KUKA KRL data list: ps_ltc_geo_c2.dat

&ACCESS RVO1
&REL 132
&COMMENT GUN C2 geom Accelo
&PARAM DISKPATH = KRC:\R1\Program\SOLDA LTC
DEFDAT  ps_ltc_geo_c2
;FOLD EXTERNAL DECLARATIONS;%{PE}%MKUKATPBASIS,%CEXT,%VCOMMON,%P
;FOLD GRIPPERTECH EXT
EXT  H50 (INT  :IN,INT  :IN,INT  :IN,GRP_TYP  :IN )
;ENDFOLD (GRIPPERTECH EXT)
;FOLD SPOTTECH EXT
EXT  USERSPOT (S_COMMAND  :IN,SPOT_TYPE  :IN )
;ENDFOLD (SPOTTECH EXT)
;FOLD BASISTECH EXT;%{PE}%MKUKATPBASIS,%CEXT,%VEXT,%P
EXT  BAS (BAS_COMMAND  :IN,REAL  :IN )
DECL INT SUCCESS
;ENDFOLD (BASISTECH EXT)
;FOLD USER EXT;%{E}%MKUKATPUSER,%CEXT,%VEXT,%P
;Make your modifications here

;ENDFOLD (USER EXT)
;ENDFOLD (EXTERNAL DECLARATIONS)
;# ============ START PATH : swp_p13050r3_ltc_geo_c2 =============
DECL FDAT Flx828={TOOL_NO 2,BASE_NO 2,IPO_FRAME #BASE,POINT2[] " "}
DECL PDAT PP_OLP7={VEL 100.0,ACC 100.0,APO_DIST 30.0,APO_MODE #CDIS}
DECL E6POS Xlx828={X 1313.89404,Y -1331.46704,Z 523.221985,A -13.1561899,B 25.8715191,C 86.3671722,S 2,T 11,E1 5636.96094,E2 0.0,E3 0.0,E4 0.0,E5 0.0,E6 0.0}
DECL FDAT Flx827={TOOL_NO 2,BASE_NO 2,IPO_FRAME #BASE,POINT2[] " "}
DECL PDAT PP_OLP8={VEL 100.0,ACC 100.0,APO_DIST 30.0,APO_MODE #CDIS}
DECL E6POS Xlx827={X 1268.92896,Y -1028.29199,Z 484.852692,A 0.744642675,B 44.8028793,C 92.9150925,S 2,T 11,E1 5636.54883,E2 0.0,E3 0.0,E4 0.0,E5 0.0,E6 0.0}
DECL FDAT Flx826={TOOL_NO 2,BASE_NO 2,IPO_FRAME #BASE,POINT2[] " "}
DECL PDAT PP_OLP9={VEL 100.0,ACC 100.0,APO_DIST 100.0,APO_MODE #CDIS}
DECL E6POS Xlx826={X 1247.14197,Y -839.330017,Z 487.233398,A 0.873326421,B 46.5667191,C 93.0090027,S 2,T 11,E1 5636.54297,E2 0.0,E3 0.0,E4 0.0,E5 0.0,E6 0.0}
DECL FDAT Fswp_60_0399={TOOL_NO 2,BASE_NO 2,IPO_FRAME #BASE,POINT2[] " "}
DECL PDAT PP_OLP10={VEL 100.0,ACC 100.0,APO_DIST 0.0}
DECL SPOT_TYPE SS_OLP1={GUN 1,PAIR #FIRST,RETR #OPN,CLO_TM 0,PGNO1 1,PRESS1 1.0,PGNO2 0,PRESS2 0.0}
DECL E6POS Xswp_60_0399={X 1474.19995,Y -844.473572,Z 743.300415,A 0.666425526,B -12.8179398,C 91.9345932,S 2,T 11,E1 5636.55713,E2 0.0,E3 0.0,E4 0.0,E5 0.0,E6 0.0}
DECL FDAT Fswp_60_0395={TOOL_NO 2,BASE_NO 2,IPO_FRAME #BASE,POINT2[] " "}
DECL PDAT PP_OLP12={VEL 100.0,ACC 100.0,APO_DIST 0.0}
DECL SPOT_TYPE SS_OLP2={GUN 1,PAIR #FIRST,RETR #OPN,CLO_TM 0,PGNO1 1,PRESS1 1.0,PGNO2 0,PRESS2 0.0}
DECL E6POS Xswp_60_0395={X 1445.07202,Y -842.604614,Z 678.067871,A 1.23996997,B -7.01102686,C 91.9965591,S 2,T 11,E1 5636.50488,E2 0.0,E3 0.0,E4 0.0,E5 0.0,E6 0.0}
DECL FDAT Flx824={TOOL_NO 2,BASE_NO 2,IPO_FRAME #BASE,POINT2[] " "}
DECL PDAT PP_OLP13={VEL 100.0,ACC 100.0,APO_DIST 100.0,APO_MODE #CDIS}
DECL E6POS Xlx824={X 1443.104,Y -839.287109,Z 639.178406,A 2.08833504,B 1.78453195,C 92.0118713,S 2,T 11,E1 5636.50488,E2 0.0,E3 0.0,E4 0.0,E5 0.0,E6 0.0}
DECL FDAT Fswp_60_0393={TOOL_NO 2,BASE_NO 2,IPO_FRAME #BASE,POINT2[] " "}
DECL PDAT PP_OLP14={VEL 100.0,ACC 100.0,APO_DIST 0.0}
DECL SPOT_TYPE SS_OLP3={GUN 1,PAIR #FIRST,RETR #OPN,CLO_TM 0,PGNO1 1,PRESS1 1.0,PGNO2 0,PRESS2 0.0}
DECL E6POS Xswp_60_0393={X 1475.52795,Y -844.253113,Z 638.954773,A -0.0227528196,B 3.38127303,C 92.2101974,S 2,T 11,E1 5636.49512,E2 0.0,E3 0.0,E4 0.0,E5 0.0,E6 0.0}
DECL FDAT Flx823={TOOL_NO 2,BASE_NO 2,IPO_FRAME #BASE,POINT2[] " "}
DECL PDAT PP_OLP16={VEL 100.0,ACC 100.0,APO_DIST 100.0,APO_MODE #CDIS}
DECL E6POS Xlx823={X 1363.30005,Y -822.437317,Z 549.010315,A 0.472675204,B 20.0343704,C 92.5931931,S 2,T 11,E1 5636.54199,E2 0.0,E3 0.0,E4 0.0,E5 0.0,E6 0.0}
DECL FDAT Flx820={TOOL_NO 2,BASE_NO 2,IPO_FRAME #BASE,POINT2[] " "}
DECL PDAT PP_OLP18={VEL 100.0,ACC 100.0,APO_DIST 100.0,APO_MODE #CDIS}
DECL E6POS Xlx820={X 1251.099,Y -1023.78699,Z 483.461304,A 0.771801889,B 44.3958397,C 93.1082611,S 2,T 11,E1 5636.50977,E2 0.0,E3 0.0,E4 0.0,E5 0.0,E6 0.0}
DECL FDAT Flx819={TOOL_NO 2,BASE_NO 2,IPO_FRAME #BASE,POINT2[] " "}
DECL PDAT PP_OLP19={VEL 100.0,ACC 100.0,APO_DIST 100.0,APO_MODE #CDIS}
DECL E6POS Xlx819={X 1444.45801,Y -1414.67004,Z 462.043915,A -12.3754196,B 44.4594803,C 91.9307175,S 2,T 11,E1 5636.50586,E2 0.0,E3 0.0,E4 0.0,E5 0.0,E6 0.0}
DECL FDAT Fswp_60_0341={TOOL_NO 2,BASE_NO 2,IPO_FRAME #BASE,POINT2[] " "}
DECL PDAT PP_OLP21={VEL 100.0,ACC 100.0,APO_DIST 0.0}
DECL SPOT_TYPE SS_OLP4={GUN 1,PAIR #FIRST,RETR #OPN,CLO_TM 0,PGNO1 1,PRESS1 1.0,PGNO2 0,PRESS2 0.0}
DECL E6POS Xswp_60_0341={X 1400.88696,Y -841.813171,Z 60.6647987,A -3.50004601,B 32.0640984,C 89.0238266,S 2,T 11,E1 5553.2959,E2 0.0,E3 0.0,E4 0.0,E5 0.0,E6 0.0}
DECL FDAT Fswp_60_0333={TOOL_NO 2,BASE_NO 2,IPO_FRAME #BASE,POINT2[] " "}
DECL PDAT PP_OLP22={VEL 100.0,ACC 100.0,APO_DIST 0.0}
DECL SPOT_TYPE SS_OLP5={GUN 1,PAIR #FIRST,RETR #OPN,CLO_TM 0,PGNO1 1,PRESS1 1.0,PGNO2 0,PRESS2 0.0}
DECL E6POS Xswp_60_0333={X 1245.823,Y -840.628174,Z 60.1122894,A -3.49715209,B 31.6406898,C 88.9972,S 2,T 11,E1 5553.13379,E2 0.0,E3 0.0,E4 0.0,E5 0.0,E6 0.0}
DECL FDAT Flx815={TOOL_NO 2,BASE_NO 2,IPO_FRAME #BASE,POINT2[] " "}
DECL PDAT PP_OLP23={VEL 100.0,ACC 100.0,APO_DIST 100.0,APO_MODE #CDIS}
DECL E6POS Xlx815={X 1196.84094,Y -826.712402,Z 159.871796,A -3.81221008,B 31.1064892,C 88.8207474,S 2,T 11,E1 5552.36182,E2 0.0,E3 0.0,E4 0.0,E5 0.0,E6 0.0}
DECL FDAT Flx816={TOOL_NO 2,BASE_NO 2,IPO_FRAME #BASE,POINT2[] " "}
DECL PDAT PP_OLP24={VEL 100.0,ACC 100.0,APO_DIST 30.0,APO_MODE #CDIS}
DECL E6POS Xlx816={X 1198.349,Y -1363.80798,Z 157.276199,A -10.3484898,B 31.0169201,C 86.4901962,S 2,T 11,E1 5539.03516,E2 0.0,E3 0.0,E4 0.0,E5 0.0,E6 0.0}
DECL FDAT Flx814={TOOL_NO 2,BASE_NO 2,IPO_FRAME #BASE,POINT2[] " "}
DECL E6POS Xlx814={X 369.932312,Y -1519.18604,Z -172.970001,A -167.901596,B 57.7843094,C -67.7142334,S 2,T 11,E1 4678.13623,E2 0.0,E3 0.0,E4 0.0,E5 0.0,E6 0.0}
DECL FDAT Flx813={TOOL_NO 2,BASE_NO 2,IPO_FRAME #BASE,POINT2[] " "}
DECL E6POS Xlx813={X 428.942688,Y -806.54657,Z -98.9288864,A 175.669601,B 53.0529213,C -91.0339203,S 2,T 11,E1 4678.10986,E2 0.0,E3 0.0,E4 0.0,E5 0.0,E6 0.0}
DECL FDAT Fswp_60_0255={TOOL_NO 2,BASE_NO 2,IPO_FRAME #BASE,POINT2[] " "}
DECL PDAT PP_OLP30={VEL 100.0,ACC 100.0,APO_DIST 0.0}
DECL SPOT_TYPE SS_OLP6={GUN 1,PAIR #FIRST,RETR #OPN,CLO_TM 0,PGNO1 1,PRESS1 1.0,PGNO2 0,PRESS2 0.0}
DECL E6POS Xswp_60_0255={X 300.463989,Y -853.163086,Z -119.2994,A 175.893997,B 45.7151489,C -93.9277267,S 2,T 11,E1 4678.07178,E2 0.0,E3 0.0,E4 0.0,E5 0.0,E6 0.0}
DECL FDAT Fswp_60_0245={TOOL_NO 2,BASE_NO 2,IPO_FRAME #BASE,POINT2[] " "}
DECL PDAT PP_OLP31={VEL 100.0,ACC 100.0,APO_DIST 0.0}
DECL SPOT_TYPE SS_OLP7={GUN 1,PAIR #FIRST,RETR #OPN,CLO_TM 0,PGNO1 1,PRESS1 1.0,PGNO2 0,PRESS2 0.0}
DECL E6POS Xswp_60_0245={X 236.971893,Y -854.070374,Z -10.8238602,A -179.4767,B 23.06007,C -91.1865311,S 2,T 11,E1 4684.35791,E2 0.0,E3 0.0,E4 0.0,E5 0.0,E6 0.0}
DECL FDAT Fswp_60_0235={TOOL_NO 2,BASE_NO 2,IPO_FRAME #BASE,POINT2[] " "}
DECL PDAT PP_OLP33={VEL 100.0,ACC 100.0,APO_DIST 0.0}
DECL SPOT_TYPE SS_OLP8={GUN 1,PAIR #FIRST,RETR #OPN,CLO_TM 0,PGNO1 1,PRESS1 1.0,PGNO2 0,PRESS2 0.0}
DECL E6POS Xswp_60_0235={X 258.574402,Y -852.900208,Z 151.175507,A -179.494904,B -23.2381096,C -89.6756897,S 2,T 11,E1 4681.46387,E2 0.0,E3 0.0,E4 0.0,E5 0.0,E6 0.0}
DECL FDAT Flx798={TOOL_NO 2,BASE_NO 2,IPO_FRAME #BASE,POINT2[] " "}
DECL PDAT PP_OLP34={VEL 100.0,ACC 100.0,APO_DIST 100.0,APO_MODE #CDIS}
DECL E6POS Xlx798={X 268.457794,Y -793.195618,Z 67.879303,A -179.860504,B 7.61739111,C -89.3985977,S 2,T 11,E1 4683.8208,E2 0.0,E3 0.0,E4 0.0,E5 0.0,E6 0.0}
DECL FDAT Flx799={TOOL_NO 2,BASE_NO 2,IPO_FRAME #BASE,POINT2[] " "}
DECL PDAT PP_OLP35={VEL 100.0,ACC 100.0,APO_DIST 100.0,APO_MODE #CDIS}
DECL E6POS Xlx799={X 345.372589,Y -812.418274,Z -84.5929871,A 176.158905,B 42.65382,C -93.2365875,S 2,T 11,E1 4677.79199,E2 0.0,E3 0.0,E4 0.0,E5 0.0,E6 0.0}
DECL FDAT Flx800={TOOL_NO 2,BASE_NO 2,IPO_FRAME #BASE,POINT2[] " "}
DECL E6POS Xlx800={X 428.928711,Y -806.551819,Z -98.9253006,A 175.669693,B 53.0524902,C -91.0339737,S 2,T 11,E1 4686.33398,E2 0.0,E3 0.0,E4 0.0,E5 0.0,E6 0.0}
DECL FDAT Flx802={TOOL_NO 2,BASE_NO 2,IPO_FRAME #BASE,POINT2[] " "}
DECL PDAT PP_OLP37={VEL 100.0,ACC 100.0,APO_DIST 100.0,APO_MODE #CDIS}
DECL E6POS Xlx802={X 410.083588,Y -1114.28699,Z -102.263397,A 175.624405,B 54.5072289,C -91.0710373,S 2,T 11,E1 4684.38477,E2 0.0,E3 0.0,E4 0.0,E5 0.0,E6 0.0}
DECL FDAT Flx801={TOOL_NO 2,BASE_NO 2,IPO_FRAME #BASE,POINT2[] " "}
DECL PDAT PP_OLP38={VEL 100.0,ACC 100.0,APO_DIST 10.0,APO_MODE #CDIS}
DECL E6POS Xlx801={X 350.765411,Y -1468.63098,Z -154.114105,A -172.531601,B 56.018959,C -75.8321533,S 2,T 11,E1 4678.13477,E2 0.0,E3 0.0,E4 0.0,E5 0.0,E6 0.0}
DECL FDAT Flx804={TOOL_NO 2,BASE_NO 2,IPO_FRAME #BASE,POINT2[] " "}
DECL E6POS Xlx804={X 395.674713,Y -813.304382,Z 335.053406,A -179.504196,B 41.2089806,C -87.9716721,S 2,T 11,E1 4687.36084,E2 0.0,E3 0.0,E4 0.0,E5 0.0,E6 0.0}
DECL FDAT Flx803={TOOL_NO 2,BASE_NO 2,IPO_FRAME #BASE,POINT2[] " "}
DECL PDAT PP_OLP45={VEL 100.0,ACC 100.0,APO_DIST 100.0,APO_MODE #CDIS}
DECL E6POS Xlx803={X 236.066498,Y -818.786377,Z 292.583099,A -179.961105,B 26.3373394,C -89.4697876,S 2,T 11,E1 4682.87988,E2 0.0,E3 0.0,E4 0.0,E5 0.0,E6 0.0}
DECL FDAT Fswp_60_0229={TOOL_NO 2,BASE_NO 2,IPO_FRAME #BASE,POINT2[] " ",TQ_STATE FALSE}
DECL PDAT PP_OLP46={VEL 100.0,ACC 100.0,APO_DIST 0.0}
DECL SPOT_TYPE SS_OLP9={GUN 1,PAIR #FIRST,RETR #OPN,CLO_TM 0,PGNO1 1,PRESS1 1.0,PGNO2 0,PRESS2 0.0}
DECL E6POS Xswp_60_0229={X 216.704895,Y -869.258728,Z 250.863495,A -179.965103,B 26.5219803,C -89.4639969,S 2,T 11,E1 4685.6792,E2 0.0,E3 0.0,E4 0.0,E5 0.0,E6 0.0}
DECL FDAT Fswp_60_0225={TOOL_NO 2,BASE_NO 2,IPO_FRAME #BASE,POINT2[] " "}
DECL PDAT PP_OLP47={VEL 100.0,ACC 100.0,APO_DIST 0.0}
DECL SPOT_TYPE SS_OLP10={GUN 1,PAIR #FIRST,RETR #OPN,CLO_TM 0,PGNO1 1,PRESS1 1.0,PGNO2 0,PRESS2 0.0}
DECL E6POS Xswp_60_0225={X 210.434692,Y -869.599915,Z 287.652191,A -178.351898,B 25.9884892,C -88.7657318,S 2,T 11,E1 4685.66895,E2 0.0,E3 0.0,E4 0.0,E5 0.0,E6 0.0}
DECL FDAT Fswp_60_0221={TOOL_NO 2,BASE_NO 2,IPO_FRAME #BASE,POINT2[] " "}
DECL PDAT PP_OLP49={VEL 100.0,ACC 100.0,APO_DIST 0.0}
DECL SPOT_TYPE SS_OLP11={GUN 1,PAIR #FIRST,RETR #OPN,CLO_TM 0,PGNO1 1,PRESS1 1.0,PGNO2 0,PRESS2 0.0}
DECL E6POS Xswp_60_0221={X 174.025696,Y -868.362915,Z 329.479706,A -177.526199,B 4.52676916,C -90.1046982,S 2,T 11,E1 4681.50488,E2 0.0,E3 0.0,E4 0.0,E5 0.0,E6 0.0}
DECL FDAT Flx795={TOOL_NO 2,BASE_NO 2,IPO_FRAME #BASE,POINT2[] " "}
DECL PDAT PP_OLP50={VEL 100.0,ACC 100.0,APO_DIST 100.0,APO_MODE #CDIS}
DECL E6POS Xlx795={X 226.200195,Y -837.525085,Z 348.480286,A -178.942001,B 2.25270796,C -89.7577896,S 2,T 11,E1 4678.92383,E2 0.0,E3 0.0,E4 0.0,E5 0.0,E6 0.0}
DECL FDAT Flx796={TOOL_NO 2,BASE_NO 2,IPO_FRAME #BASE,POINT2[] " "}
DECL PDAT PP_OLP51={VEL 100.0,ACC 100.0,APO_DIST 100.0,APO_MODE #CDIS}
DECL E6POS Xlx796={X 263.717407,Y -815.125122,Z 435.898987,A -178.984207,B 0.893851578,C -89.7701492,S 2,T 11,E1 4682.00098,E2 0.0,E3 0.0,E4 0.0,E5 0.0,E6 0.0}
DECL FDAT Fswp_60_0205={TOOL_NO 2,BASE_NO 2,IPO_FRAME #BASE,POINT2[] " "}
DECL PDAT PP_OLP52={VEL 100.0,ACC 100.0,APO_DIST 0.0}
DECL SPOT_TYPE SS_OLP12={GUN 1,PAIR #FIRST,RETR #OPN,CLO_TM 0,PGNO1 1,PRESS1 1.0,PGNO2 0,PRESS2 0.0}
DECL E6POS Xswp_60_0205={X 265.348785,Y -866.557007,Z 493.816589,A -178.943497,B 1.47540104,C -89.7626266,S 2,T 11,E1 4677.98193,E2 0.0,E3 0.0,E4 0.0,E5 0.0,E6 0.0}
DECL FDAT Fswp_60_0209={TOOL_NO 2,BASE_NO 2,IPO_FRAME #BASE,POINT2[] " "}
DECL SPOT_TYPE SS_OLP13={GUN 1,PAIR #FIRST,RETR #OPN,CLO_TM 0,PGNO1 1,PRESS1 1.0,PGNO2 0,PRESS2 0.0}
DECL E6POS Xswp_60_0209={X 198.4814,Y -864.90863,Z 453.328186,A -179.031296,B -7.38044596,C -89.7764587,S 2,T 11,E1 4674.09521,E2 0.0,E3 0.0,E4 0.0,E5 0.0,E6 0.0}
DECL FDAT Fswp_60_0217={TOOL_NO 2,BASE_NO 2,IPO_FRAME #BASE,POINT2[] " "}
DECL SPOT_TYPE SS_OLP14={GUN 1,PAIR #FIRST,RETR #OPN,CLO_TM 0,PGNO1 1,PRESS1 1.0,PGNO2 0,PRESS2 0.0}
DECL E6POS Xswp_60_0217={X 129.435394,Y -861.487915,Z 279.004608,A 17.8512707,B -39.6672592,C 83.1958389,S 2,T 11,E1 4906.23389,E2 0.0,E3 0.0,E4 0.0,E5 0.0,E6 0.0}
DECL FDAT Fswp_60_0219={TOOL_NO 2,BASE_NO 2,IPO_FRAME #BASE,POINT2[] " "}
DECL SPOT_TYPE SS_OLP15={GUN 1,PAIR #FIRST,RETR #OPN,CLO_TM 0,PGNO1 1,PRESS1 1.0,PGNO2 0,PRESS2 0.0}
DECL E6POS Xswp_60_0219={X 132.783798,Y -863.262512,Z 297.808594,A 16.7955704,B -40.7878494,C 86.3009567,S 2,T 11,E1 4905.89502,E2 0.0,E3 0.0,E4 0.0,E5 0.0,E6 0.0}
DECL FDAT Flx780={TOOL_NO 2,BASE_NO 2,IPO_FRAME #BASE,POINT2[] " "}
DECL PDAT PP_OLP71={VEL 100.0,ACC 100.0,APO_DIST 25.0,APO_MODE #CDIS}
DECL E6POS Xlx780={X -536.1073,Y -3036.90088,Z -433.383789,A -103.127502,B 3.39632702,C 10.3325796,S 2,T 11,E1 3967.95703,E2 0.0,E3 0.0,E4 0.0,E5 0.0,E6 0.0}
DECL FDAT Fswp_60_0201={TOOL_NO 2,BASE_NO 2,IPO_FRAME #BASE,POINT2[] " "}
DECL SPOT_TYPE SS_OLP16={GUN 1,PAIR #FIRST,RETR #OPN,CLO_TM 0,PGNO1 1,PRESS1 1.0,PGNO2 0,PRESS2 0.0}
DECL E6POS Xswp_60_0201={X 229.770004,Y -890.145325,Z 555.893982,A -179.049301,B -22.7869892,C -89.742157,S 2,T 11,E1 4680.5332,E2 0.0,E3 0.0,E4 0.0,E5 0.0,E6 0.0}
DECL FDAT Flx767={TOOL_NO 2,BASE_NO 2,IPO_FRAME #BASE,POINT2[] " "}
DECL PDAT PP_OLP81={VEL 100.0,ACC 100.0,APO_DIST 30.0,APO_MODE #CDIS}
DECL E6POS Xlx767={X -4198.59521,Y -2862.68604,Z -364.78479,A 103.820503,B 2.44905901,C -6.20870399,S 2,T 43,E1 1408.61401,E2 0.0,E3 0.0,E4 0.0,E5 0.0,E6 0.0}
DECL BASIS_SUGG_T LAST_BASIS={POINT1[] "PS01010001              ",POINT2[] "PS01010001              ",CP_PARAMS[] "CPDAT0                  ",PTP_PARAMS[] "PDAT0                   ",CONT[] "                        ",CP_VEL[] "2.0                     ",PTP_VEL[] "100                     ",SPL_NAME[] "S0                      "}
DECL E6POS XP2={X -483.254089,Y -2982.05591,Z -402.20639,A -107.179497,B 0.544633925,C 4.32910204,S 2,T 3,E1 4351.56006,E2 0.0,E3 0.0,E4 0.0,E5 0.0,E6 0.0}
DECL FDAT FP2={TOOL_NO 2,BASE_NO 2,IPO_FRAME #BASE,POINT2[] " ",TQ_STATE FALSE}
DECL PDAT PPDAT2={VEL 100.0,ACC 100.0,APO_DIST 30.0,APO_MODE #CDIS}
DECL SPOT_SUGG_T LAST_SPOT={GUN[] "2                       ",RETR_CMD[] "#OPN                    ",CHOISE[] "#FIRST                  ",CLO_TM[] "1                       ",PGNO1[] "252                     ",PRESS1[] "0                       ",PGNO2[] "1                       ",PRESS2[] "0                       ",SPOT_PARAMS[] "NORMAL                  "}
DECL E6POS XP6={X 1279.60999,Y -1373.32605,Z 198.834396,A -9.93967724,B 7.73596001,C 90.3461227,S 2,T 11,E1 5553.88281,E2 0.0,E3 0.0,E4 0.0,E5 0.0,E6 0.0}
DECL FDAT FP6={TOOL_NO 2,BASE_NO 2,IPO_FRAME #BASE,POINT2[] " ",TQ_STATE FALSE}
DECL PDAT PPDAT6={VEL 100.0,ACC 100.0,APO_DIST 30.0,APO_MODE #CDIS}
DECL E6POS XP7={X 1202.75,Y -808.4328,Z 199.5867,A -5.53556919,B 7.68426991,C 92.4831314,S 2,T 11,E1 5553.88184,E2 0.0,E3 0.0,E4 0.0,E5 0.0,E6 0.0}
DECL FDAT FP7={TOOL_NO 2,BASE_NO 2,IPO_FRAME #BASE,POINT2[] " ",TQ_STATE FALSE}
DECL PDAT PPDAT7={VEL 100.0,ACC 100.0,APO_DIST 100.0}
DECL E6POS XP11={X 262.014008,Y -846.799622,Z 144.059601,A -179.474792,B -23.1920395,C -89.2290115,S 2,T 11,E1 4682.82422,E2 0.0,E3 0.0,E4 0.0,E5 0.0,E6 0.0}
DECL FDAT FP11={TOOL_NO 2,BASE_NO 2,IPO_FRAME #BASE,POINT2[] " ",TQ_STATE FALSE}
DECL PDAT PPDAT11={VEL 100.0,ACC 100.0,APO_DIST 10.0,APO_MODE #CDIS}
DECL LDAT LCPDAT1={VEL 2.0,ACC 100.0,APO_DIST 2.0,APO_FAC 50.0,AXIS_VEL 100.0,AXIS_ACC 100.0,ORI_TYP #VAR,CIRC_TYP #BASE,JERK_FAC 50.0,GEAR_JERK 50.0,EXAX_IGN 0}
DECL LDAT LCPDAT5={VEL 2.0,ACC 100.0,APO_DIST 20.0,APO_FAC 50.0,AXIS_VEL 100.0,AXIS_ACC 100.0,ORI_TYP #VAR,CIRC_TYP #BASE,JERK_FAC 50.0,GEAR_JERK 50.0,EXAX_IGN 0}
DECL LDAT LCPDAT8={VEL 2.0,ACC 100.0,APO_DIST 2.0,APO_FAC 50.0,AXIS_VEL 100.0,AXIS_ACC 100.0,ORI_TYP #VAR,CIRC_TYP #BASE,JERK_FAC 50.0,GEAR_JERK 50.0,EXAX_IGN 0}
DECL E6POS XP28={X 680.9328,Y -2572.68799,Z -141.916397,A -67.8898773,B 12.2103901,C 37.8295212,S 2,T 11,E1 4582.3208,E2 0.0,E3 0.0,E4 0.0,E5 0.0,E6 0.0}
DECL FDAT FP28={TOOL_NO 2,BASE_NO 2,IPO_FRAME #BASE,POINT2[] " ",TQ_STATE FALSE}
DECL PDAT PPDAT28={VEL 100.0,ACC 100.0,APO_DIST 100.0,APO_MODE #CDIS}
DECL E6POS XP30={X 1907.59802,Y -7875.57715,Z 2378.80493,A -86.6201935,B -16.2818298,C 91.4838104,S 2,T 11,E1 5636.49512,E2 0.0,E3 0.0,E4 0.0,E5 0.0,E6 0.0}
DECL FDAT FP30={TOOL_NO 2,BASE_NO 0,IPO_FRAME #BASE,POINT2[] " ",TQ_STATE FALSE}
DECL PDAT PPDAT30={VEL 100.0,ACC 100.0,APO_DIST 20.0,APO_MODE #CDIS}
DECL PDAT PPDAT35={VEL 100.0,ACC 100.0,APO_DIST 10.0,APO_MODE #CDIS}
DECL E6POS XP35={X -142.686005,Y -2282.2041,Z 1278.44495,A 13.8204603,B 2.44905901,C -6.20870399,S 2,T 43,E1 1408.61401,E2 0.0,E3 0.0,E4 0.0,E5 0.0,E6 0.0}
DECL FDAT FP35={TOOL_NO 2,BASE_NO 0,IPO_FRAME #BASE,POINT2[] " ",TQ_STATE FALSE}
DECL PDAT PPDAT36={VEL 100.0,ACC 100.0,APO_DIST 5.0,APO_MODE #CDIS}
DECL E6POS XP36={X -694.74707,Y -860.123779,Z 1278.44604,A -105.193901,B 2.44900703,C -6.20870686,S 2,T 42,E1 1408.61401,E2 0.0,E3 0.0,E4 0.0,E5 0.0,E6 0.0}
DECL FDAT FP36={TOOL_NO 2,BASE_NO 0,IPO_FRAME #BASE,POINT2[] " ",TQ_STATE FALSE}
DECL PDAT PPDAT37={VEL 100.0,ACC 100.0,APO_DIST 5.0,APO_MODE #CDIS}
DECL E6POS Xswp_60_0337={X 1321.69104,Y -841.830078,Z 60.7148399,A -3.494941,B 32.0055504,C 89.0259399,S 2,T 11,E1 5553.2749,E2 0.0,E3 0.0,E4 0.0,E5 0.0,E6 0.0}
DECL FDAT Fswp_60_0337={TOOL_NO 2,BASE_NO 2,IPO_FRAME #BASE,POINT2[] " ",TQ_STATE FALSE}
DECL E6POS XP37={X 240.859299,Y 679.959473,Z 1415.14001,A -41.8363991,B 11.3211298,C 18.1852207,S 2,T 2,E1 1820.02405,E2 0.0,E3 0.0,E4 0.0,E5 0.0,E6 0.0}
DECL FDAT FP37={TOOL_NO 2,BASE_NO 0,IPO_FRAME #BASE,POINT2[] " ",TQ_STATE FALSE}
DECL PDAT PPDAT38={VEL 100.0,ACC 100.0,APO_DIST 100.0,APO_MODE #CDIS}
DECL E6POS XP41={X 1435.64795,Y -841.162292,Z 747.776978,A 1.34821701,B -15.5304098,C 91.8447266,S 2,T 11,E1 5636.5,E2 0.0,E3 0.0,E4 0.0,E5 0.0,E6 0.0}
DECL FDAT FP41={TOOL_NO 2,BASE_NO 2,IPO_FRAME #BASE,POINT2[] " ",TQ_STATE FALSE}
DECL PDAT PPDAT42={VEL 100.0,ACC 100.0,APO_DIST 5.0,APO_MODE #CDIS}
DECL E6POS XP42={X 1251.14099,Y -838.862915,Z 486.759308,A 0.970713615,B 46.9011612,C 93.2508469,S 2,T 11,E1 5636.50684,E2 0.0,E3 0.0,E4 0.0,E5 0.0,E6 0.0}
DECL FDAT FP42={TOOL_NO 2,BASE_NO 2,IPO_FRAME #BASE,POINT2[] " ",TQ_STATE FALSE}
DECL PDAT PPDAT43={VEL 100.0,ACC 100.0,APO_DIST 3.0,APO_MODE #CDIS}
DECL E6POS XP43={X 389.176086,Y -1114.28699,Z -102.269798,A 175.624603,B 54.5074883,C -91.0707474,S 2,T 11,E1 4678.20117,E2 0.0,E3 0.0,E4 0.0,E5 0.0,E6 0.0}
DECL FDAT FP43={TOOL_NO 2,BASE_NO 2,IPO_FRAME #BASE,POINT2[] " ",TQ_STATE FALSE}
DECL PDAT PP_OLP84={VEL 100.0,ACC 100.0,APO_DIST 0.0}
DECL E6POS XP47={X -5620.67822,Y -3414.75,Z -364.782715,A -15.1935997,B 2.44905591,C -6.20877123,S 2,T 42,E1 1408.61401,E2 0.0,E3 0.0,E4 0.0,E5 0.0,E6 0.0}
DECL FDAT FP47={TOOL_NO 2,BASE_NO 2,IPO_FRAME #BASE,POINT2[] " ",TQ_STATE FALSE}
DECL PDAT PPDAT51={VEL 100.0,ACC 100.0,APO_DIST 5.0,APO_MODE #CDIS}
DECL PDAT PPDAT55={VEL 100.0,ACC 100.0,APO_DIST 100.0}
DECL PDAT PPDAT56={VEL 100.0,ACC 100.0,APO_DIST 100.0}
DECL PDAT PPDAT57={VEL 100.0,ACC 100.0,APO_DIST 100.0}
DECL PDAT PPDAT58={VEL 100.0,ACC 100.0,APO_DIST 100.0}
DECL E6POS XP50={X 269.843292,Y -848.116577,Z 60.8358002,A -179.496094,B 10.1010799,C -90.1158066,S 2,T 11,E1 4681.69385,E2 0.0,E3 0.0,E4 0.0,E5 0.0,E6 0.0}
DECL FDAT FP50={TOOL_NO 2,BASE_NO 2,IPO_FRAME #BASE,POINT2[] " ",TQ_STATE FALSE}
DECL PDAT PPDAT59={VEL 100.0,ACC 100.0,APO_DIST 10.0,APO_MODE #CDIS}
DECL PDAT PPDAT60={VEL 100.0,ACC 100.0,APO_DIST 100.0}
DECL PDAT PPDAT61={VEL 100.0,ACC 100.0,APO_DIST 100.0}
DECL PDAT PPDAT62={VEL 100.0,ACC 100.0,APO_DIST 100.0}
DECL PDAT PPDAT63={VEL 100.0,ACC 100.0,APO_DIST 100.0}
DECL E6POS XP51={X 278.781891,Y -850.64032,Z 529.158386,A -179.048996,B -22.7865505,C -89.7425766,S 2,T 11,E1 4682.99902,E2 0.0,E3 0.0,E4 0.0,E5 0.0,E6 0.0}
DECL FDAT FP51={TOOL_NO 2,BASE_NO 2,IPO_FRAME #BASE,POINT2[] " ",TQ_STATE FALSE}
DECL PDAT PPDAT65={VEL 100.0,ACC 100.0,APO_DIST 20.0,APO_MODE #CDIS}
DECL E6POS XP53={X 342.528687,Y -1312.19995,Z 567.050598,A 179.099304,B -30.7727299,C -90.2307968,S 2,T 11,E1 4679.25,E2 0.0,E3 0.0,E4 0.0,E5 0.0,E6 0.0}
DECL FDAT FP53={TOOL_NO 2,BASE_NO 2,IPO_FRAME #BASE,POINT2[] " ",TQ_STATE FALSE}
DECL PDAT PPDAT67={VEL 100.0,ACC 100.0,APO_DIST 100.0,APO_MODE #CDIS}
DECL PDAT PPDAT0={VEL 100.0,ACC 100.0,APO_DIST 100.0,APO_MODE #CDIS}
DECL E6POS XP0={X 496.141388,Y -1715.23999,Z -107.852203,A -18.1212292,B -8.07049656,C 74.2473679,S 2,T 11,E1 4684.875,E2 0.0,E3 0.0,E4 0.0,E5 0.0,E6 0.0}
DECL FDAT FP0={TOOL_NO 2,BASE_NO 2,IPO_FRAME #BASE,POINT2[] " ",TQ_STATE FALSE}
DECL PDAT PPDAT69={VEL 100.0,ACC 100.0,APO_DIST 100.0,APO_MODE #CDIS}
DECL E6POS XP55={X -33.49963,Y -879.133728,Z 149.150299,A 18.1609402,B -38.4940681,C 79.5255966,S 2,T 11,E1 4860.08496,E2 0.0,E3 0.0,E4 0.0,E5 0.0,E6 0.0}
DECL FDAT FP55={TOOL_NO 2,BASE_NO 2,IPO_FRAME #BASE,POINT2[] " ",TQ_STATE FALSE}
DECL PDAT PPDAT70={VEL 100.0,ACC 100.0,APO_DIST 30.0,APO_MODE #CDIS}
DECL E6POS XP56={X 99.2140808,Y -846.499817,Z 258.782196,A 18.1166897,B -38.3201714,C 79.6072464,S 2,T 11,E1 4902.61377,E2 0.0,E3 0.0,E4 0.0,E5 0.0,E6 0.0}
DECL FDAT FP56={TOOL_NO 2,BASE_NO 2,IPO_FRAME #BASE,POINT2[] " ",TQ_STATE FALSE}
DECL PDAT PPDAT71={VEL 100.0,ACC 100.0,APO_DIST 100.0,APO_MODE #CDIS}
DECL E6POS XP57={X 107.837502,Y -825.859619,Z 258.730988,A 18.1646595,B -38.4922714,C 79.5321808,S 2,T 11,E1 4907.47314,E2 0.0,E3 0.0,E4 0.0,E5 0.0,E6 0.0}
DECL FDAT FP57={TOOL_NO 2,BASE_NO 2,IPO_FRAME #BASE,POINT2[] " ",TQ_STATE FALSE}
DECL PDAT PP_OLP86={VEL 100.0,ACC 100.0,APO_DIST 0.0}
DECL PDAT PP_OLP87={VEL 100.0,ACC 100.0,APO_DIST 0.0}
DECL PDAT PP_OLP88={VEL 100.0,ACC 100.0,APO_DIST 100.0,APO_MODE #CDIS}
DECL E6POS Xlx788={X 106.594398,Y -825.886902,Z 270.356812,A 18.1619492,B -38.495739,C 79.5243073,S 2,T 11,E1 4905.55518,E2 0.0,E3 0.0,E4 0.0,E5 0.0,E6 0.0}
DECL FDAT Flx788={TOOL_NO 2,BASE_NO 2,IPO_FRAME #BASE,POINT2[] " "}
DECL PDAT PP_OLP89={VEL 100.0,ACC 100.0,APO_DIST 100.0,APO_MODE #CDIS}
DECL E6POS Xlx831={X -33.5169907,Y -895.781006,Z 149.145905,A 18.1617107,B -38.4911385,C 79.5256271,S 2,T 11,E1 4900.61523,E2 0.0,E3 0.0,E4 0.0,E5 0.0,E6 0.0}
DECL FDAT Flx831={TOOL_NO 2,BASE_NO 2,IPO_FRAME #BASE,POINT2[] " "}
DECL E6POS XP59={X 496.141388,Y -1715.23999,Z -107.852203,A -18.1212292,B -8.07049656,C 74.2473679,S 2,T 11,E1 4684.875,E2 0.0,E3 0.0,E4 0.0,E5 0.0,E6 0.0}
DECL FDAT FP59={TOOL_NO 2,BASE_NO 2,IPO_FRAME #BASE,POINT2[] " ",TQ_STATE FALSE}
DECL PDAT PPDAT73={VEL 100.0,ACC 100.0,APO_DIST 100.0,APO_MODE #CDIS}
DECL E6POS XP62={X 390.037506,Y -1524.04297,Z 353.998199,A -179.504196,B 41.2089806,C -87.9716721,S 2,T 11,E1 4687.36084,E2 0.0,E3 0.0,E4 0.0,E5 0.0,E6 0.0}
DECL FDAT FP62={TOOL_NO 2,BASE_NO 2,IPO_FRAME #BASE,POINT2[] " ",TQ_STATE FALSE}
DECL LDAT LCPDAT11={VEL 2.0,ACC 80.0,APO_DIST 20.0,APO_FAC 50.0,AXIS_VEL 100.0,AXIS_ACC 100.0,ORI_TYP #VAR,CIRC_TYP #BASE,JERK_FAC 50.0,GEAR_JERK 50.0,EXAX_IGN 0}
DECL PDAT PPDAT76={VEL 100.0,ACC 100.0,APO_DIST 100.0}
DECL PDAT PP_OLP91={VEL 100.0,ACC 100.0,APO_DIST 0.0}
DECL E6POS Xswp_60_0203={X 258.56131,Y -891.100525,Z 551.157715,A -179.048798,B -22.7876396,C -89.7420273,S 2,T 11,E1 4680.53418,E2 0.0,E3 0.0,E4 0.0,E5 0.0,E6 0.0}
DECL FDAT Fswp_60_0203={TOOL_NO 2,BASE_NO 2,IPO_FRAME #BASE,POINT2[] " "}
DECL PDAT PPDAT77={VEL 100.0,ACC 100.0,APO_DIST 5.0,APO_MODE #CDIS}
DECL E6POS XP63={X 278.777405,Y -824.098328,Z 529.155823,A -179.048904,B -22.7866707,C -89.7424927,S 2,T 11,E1 4679.38281,E2 0.0,E3 0.0,E4 0.0,E5 0.0,E6 0.0}
DECL FDAT FP63={TOOL_NO 2,BASE_NO 2,IPO_FRAME #BASE,POINT2[] " ",TQ_STATE FALSE}
DECL PDAT PPDAT78={VEL 100.0,ACC 100.0,APO_DIST 5.0,APO_MODE #CDIS}
DECL E6POS XP64={X 362.55191,Y -821.745605,Z 567.791321,A 178.825394,B -34.4097099,C -89.7091599,S 2,T 43,E1 4681.0,E2 0.0,E3 0.0,E4 0.0,E5 0.0,E6 0.0}
DECL FDAT FP64={TOOL_NO 2,BASE_NO 2,IPO_FRAME #BASE,POINT2[] " ",TQ_STATE FALSE}
DECL PDAT PPDAT81={VEL 50.0,ACC 100.0,APO_DIST 100.0}
DECL PDAT PPDAT82={VEL 50.0,ACC 100.0,APO_DIST 100.0}
DECL PDAT PPDAT83={VEL 50.0,ACC 100.0,APO_DIST 100.0}
DECL PDAT PPDAT84={VEL 50.0,ACC 100.0,APO_DIST 100.0}
DECL E6POS Xswp_60_0259={X 366.820313,Y -853.075012,Z -120.775597,A 174.980896,B 53.6071014,C -94.6270599,S 2,T 11,E1 4678.04688,E2 0.0,E3 0.0,E4 0.0,E5 0.0,E6 0.0}
DECL FDAT Fswp_60_0259={TOOL_NO 2,BASE_NO 2,IPO_FRAME #BASE,POINT2[] " ",TQ_STATE FALSE}
DECL E6POS Xswp_60_0253={X 259.621399,Y -852.773804,Z -112.924301,A -178.049194,B 45.6860199,C -87.9386673,S 2,T 11,E1 4677.8291,E2 0.0,E3 0.0,E4 0.0,E5 0.0,E6 0.0}
DECL FDAT Fswp_60_0253={TOOL_NO 2,BASE_NO 2,IPO_FRAME #BASE,POINT2[] " ",TQ_STATE FALSE}
DECL E6POS Xswp_60_0249={X 214.160507,Y -853.164429,Z -78.3120117,A -178.291702,B 37.4617691,C -88.298378,S 2,T 11,E1 4677.83301,E2 0.0,E3 0.0,E4 0.0,E5 0.0,E6 0.0}
DECL FDAT Fswp_60_0249={TOOL_NO 2,BASE_NO 2,IPO_FRAME #BASE,POINT2[] " ",TQ_STATE FALSE}
DECL E6POS Xswp_60_0241={X 257.142303,Y -852.976929,Z 45.2910118,A -179.496002,B 10.1006603,C -90.1179733,S 2,T 11,E1 4681.69678,E2 0.0,E3 0.0,E4 0.0,E5 0.0,E6 0.0}
DECL FDAT Fswp_60_0241={TOOL_NO 2,BASE_NO 2,IPO_FRAME #BASE,POINT2[] " ",TQ_STATE FALSE}
DECL E6POS Xswp_60_0239={X 265.541687,Y -851.06073,Z 82.2472382,A -179.690903,B 4.42705202,C -90.1465073,S 2,T 11,E1 4681.69385,E2 0.0,E3 0.0,E4 0.0,E5 0.0,E6 0.0}
DECL FDAT Fswp_60_0239={TOOL_NO 2,BASE_NO 2,IPO_FRAME #BASE,POINT2[] " ",TQ_STATE FALSE}
DECL E6POS Xswp_60_0237={X 262.622711,Y -853.462097,Z 116.181099,A -179.442596,B -10.01577,C -89.6991882,S 2,T 11,E1 4682.28613,E2 0.0,E3 0.0,E4 0.0,E5 0.0,E6 0.0}
DECL FDAT Fswp_60_0237={TOOL_NO 2,BASE_NO 2,IPO_FRAME #BASE,POINT2[] " ",TQ_STATE FALSE}
DECL E6POS Xswp_60_0207={X 224.656998,Y -864.158813,Z 450.397491,A -179.030899,B -7.38146114,C -89.7758408,S 2,T 11,E1 4674.09619,E2 0.0,E3 0.0,E4 0.0,E5 0.0,E6 0.0}
DECL FDAT Fswp_60_0207={TOOL_NO 2,BASE_NO 2,IPO_FRAME #BASE,POINT2[] " ",TQ_STATE FALSE}
DECL E6POS Xswp_60_0211={X 171.593903,Y -861.216125,Z 453.690796,A -175.8172,B -7.38104677,C -89.7739334,S 2,T 11,E1 4674.09082,E2 0.0,E3 0.0,E4 0.0,E5 0.0,E6 0.0}
DECL FDAT Fswp_60_0211={TOOL_NO 2,BASE_NO 2,IPO_FRAME #BASE,POINT2[] " ",TQ_STATE FALSE}
DECL E6POS Xswp_60_0331={X 1214.06104,Y -841.564575,Z 58.9755516,A -1.34586596,B 31.1367798,C 88.9882202,S 2,T 11,E1 5552.93701,E2 0.0,E3 0.0,E4 0.0,E5 0.0,E6 0.0}
DECL FDAT Fswp_60_0331={TOOL_NO 2,BASE_NO 2,IPO_FRAME #BASE,POINT2[] " ",TQ_STATE FALSE}
DECL E6POS Xswp_60_0335={X 1281.28101,Y -841.706726,Z 60.742691,A -3.49542499,B 32.0074692,C 89.0247269,S 2,T 11,E1 5553.27783,E2 0.0,E3 0.0,E4 0.0,E5 0.0,E6 0.0}
DECL FDAT Fswp_60_0335={TOOL_NO 2,BASE_NO 2,IPO_FRAME #BASE,POINT2[] " ",TQ_STATE FALSE}
DECL E6POS Xswp_60_0339={X 1361.61902,Y -841.998718,Z 60.770359,A -3.49538493,B 32.0599518,C 89.028511,S 2,T 11,E1 5553.29883,E2 0.0,E3 0.0,E4 0.0,E5 0.0,E6 0.0}
DECL FDAT Fswp_60_0339={TOOL_NO 2,BASE_NO 2,IPO_FRAME #BASE,POINT2[] " ",TQ_STATE FALSE}
DECL PDAT PPDAT85={VEL 100.0,ACC 80.0,APO_DIST 5.0,APO_MODE #CDIS}
DECL E6POS XPS01010021={X 206.647995,Y -857.749084,Z 303.772003,A -178.132095,B 18.9228992,C -88.8315735,S 2,T 11,E1 4677.62793,E2 0.0,E3 0.0,E4 0.0,E5 0.0,E6 0.0}
DECL FDAT FPS01010021={TOOL_NO 2,BASE_NO 2,IPO_FRAME #BASE,POINT2[] " ",TQ_STATE FALSE}
DECL PDAT PPDAT86={VEL 100.0,ACC 100.0,APO_DIST 100.0}
DECL PDAT PP_OLP15={VEL 100.0,ACC 100.0,APO_DIST 0.0}
DECL E6POS Xswp_60_0396={X 1445.07202,Y -842.604614,Z 678.067871,A 1.23996997,B -7.01102686,C 91.9965591,S 2,T 11,E1 5636.50488,E2 0.0,E3 0.0,E4 0.0,E5 0.0,E6 0.0}
DECL FDAT Fswp_60_0396={TOOL_NO 2,BASE_NO 2,IPO_FRAME #BASE,POINT2[] " "}
DECL E6POS Xswp_60_0397={X 1444.36096,Y -846.166809,Z 702.064514,A 1.278198,B -9.91316891,C 91.9447021,S 2,T 11,E1 5636.50293,E2 0.0,E3 0.0,E4 0.0,E5 0.0,E6 0.0}
DECL FDAT Fswp_60_0397={TOOL_NO 2,BASE_NO 2,IPO_FRAME #BASE,POINT2[] " ",TQ_STATE FALSE}
DECL PDAT PP_OLP17={VEL 100.0,ACC 100.0,APO_DIST 0.0}
DECL E6POS Xswp_60_0394={X 1475.52795,Y -844.253113,Z 638.954773,A -0.0227528196,B 3.38127303,C 92.2101974,S 2,T 11,E1 5636.49512,E2 0.0,E3 0.0,E4 0.0,E5 0.0,E6 0.0}
DECL FDAT Fswp_60_0394={TOOL_NO 2,BASE_NO 2,IPO_FRAME #BASE,POINT2[] " "}
DECL E6POS Xswp_60_0391={X 1487.88794,Y -844.258911,Z 638.209717,A -0.0223123208,B 3.38131499,C 92.2097168,S 2,T 11,E1 5636.49512,E2 0.0,E3 0.0,E4 0.0,E5 0.0,E6 0.0}
DECL FDAT Fswp_60_0391={TOOL_NO 2,BASE_NO 2,IPO_FRAME #BASE,POINT2[] " ",TQ_STATE FALSE}
ENDDAT
